(*
SPDX-FileCopyrightText: © 2026 Oleksandr Tiutyk <trofimich@gmail.com>
SPDX-License-Identifier: MIT
License: https://opensource.org/license/mit
*)

(*!
<summary>
Sample activity that steps integer XPosition and YPosition workflow variables toward configured coordinates.
</summary>
<description>
Advances each coordinate by one unit per timer interval until both reach ToXPosition and ToYPosition. Supports
suspension with remaining-time preservation, cancellation, resetting and failure timer cleanup.
</description>
*)

{attribute 'no_explicit_call' := 'do not call this function block directly'}
{attribute 'enable_dynamic_creation'}
FUNCTION_BLOCK MoveFromToActivity EXTENDS TOF_Workflow.Activity IMPLEMENTS IMoveFromToActivity
VAR_STAT
	{attribute 'hide'} 
	_ClassName : STRING := __POUNAME();
END_VAR
VAR
	_ToXPosition : INT;
	_ToYPosition : INT;
	
	_PositionChangeTimer : TOF_Timers.Timer("PositionChangeTimer");
	//! <summary>Time left before the next position step, captured when suspension begins.</summary>
	_RemainingPositionChangeTime : TIME;
END_VAR
VAR CONSTANT
	//! <summary>Delay before the first position step and between subsequent steps; suspended time is excluded.</summary>
	POSITION_CHANGE_TIMER_INTERVAL : TIME := T#10MS;
END_VAR

(*!
<summary>Gets the runtime class name of this object.</summary>
*)
{attribute 'monitoring' := 'call'}
PROPERTY ClassName : REFERENCE TO STRING
GET
ClassName REF= _ClassName;
END_GET
END_PROPERTY

(*!
<summary>Sets the target integer X and Y coordinates for the activity.</summary>
<param name="toXPosition">Target X coordinate.</param>
<param name="toYPosition">Target Y coordinate.</param>
*)
METHOD Configure
VAR_INPUT
	toXPosition : INT;
	toYPosition : INT;
END_VAR
_ToXPosition := toXPosition;
_ToYPosition := toYPosition;
END_METHOD

(*!
<summary>Gets the namespace name of this object.</summary>
*)
{attribute 'monitoring' := 'call'}
PROPERTY NamespaceName : REFERENCE TO STRING
GET
NamespaceName REF= CurrentNamespace.Name;
END_GET
END_PROPERTY

(*!
<summary>Stops the position-change timer and clears saved remaining time when the activity fails.</summary>
<param name="exception">Exception that caused the failure.</param>
*)
METHOD PROTECTED OnFail
VAR_INPUT
	exception : TOF_Core.IException;
END_VAR
_RemainingPositionChangeTime := TOF_Core.Times.MIN_VALUE;

IF _PositionChangeTimer.State.Running THEN
	_PositionChangeTimer.Cancel();
	_PositionChangeTimer.Execute();
END_IF
END_METHOD

(*!
<summary>Stops the position-change timer and clears saved remaining time during resetting.</summary>
<param name="startResetting">TRUE on the initial RequestReset call; FALSE on subsequent Execute cycles.</param>
*)
METHOD PROTECTED OnResetting : TOF_Workflow.ACTIVITY_RESETTING_STATE
VAR_INPUT
	startResetting : BOOL;
END_VAR
_RemainingPositionChangeTime := TOF_Core.Times.MIN_VALUE;

IF _PositionChangeTimer.State.Running THEN
	_PositionChangeTimer.Cancel();
	_PositionChangeTimer.Execute();
END_IF

IF NOT _PositionChangeTimer.State.Running THEN
	OnResetting := TOF_Workflow.ACTIVITY_RESETTING_STATE.WORK_RESET;
END_IF
END_METHOD

(*!
<summary>Moves each coordinate by one unit after each position-change interval.</summary>
<description>
A fresh run restarts the timer with the full interval; resuming restarts it with the remaining time captured
by OnStopping, excluding suspended time. After a resumed step, subsequent steps use the full interval again.
An elapsed interval advances at most one step per call; missed intervals are not replayed. A refused timer
restart returns WORK_HALTED with a diagnostic, preserving any coordinate changes already made. Variable lookup
and conversion exceptions propagate to the activity's failure handling. The activity owner drives these
callbacks sequentially; they do not drive the activity recursively.
</description>
<param name="startRunning">Begins a fresh run, including reuse after an earlier run.</param>
<param name="startResuming">Resumes the remaining interval saved during suspension.</param>
<param name="haltReason">Describes a refused timer restart when WORK_HALTED is returned.</param>
*)
METHOD PROTECTED OnRunning : TOF_Workflow.ACTIVITY_RUNNING_STATE
VAR_INPUT
	startRunning : BOOL;
	startResuming : BOOL;
END_VAR
VAR_OUTPUT
	haltReason : WSTRING(255);
END_VAR
VAR
	xPosition : TOF_Core.GENERIC_VALUE;
	yPosition : TOF_Core.GENERIC_VALUE;

	currentXPosition : INT;
	currentYPosition : INT;
	
END_VAR
IF startRunning THEN
	IF NOT _PositionChangeTimer.SetIntervalAndRestart(interval := POSITION_CHANGE_TIMER_INTERVAL) THEN
		haltReason := "Could not start the position-change timer";
		OnRunning := TOF_Workflow.ACTIVITY_RUNNING_STATE.WORK_HALTED;
	END_IF
ELSIF startResuming THEN
	IF NOT _PositionChangeTimer.SetIntervalAndRestart(interval := _RemainingPositionChangeTime) THEN
		haltReason := "Could not resume the position-change timer";
		OnRunning := TOF_Workflow.ACTIVITY_RUNNING_STATE.WORK_HALTED;
	END_IF
ELSE
	_PositionChangeTimer.Execute();

	IF _PositionChangeTimer.Elapsed THEN
		IF NOT TryGetVariable(name := 'XPosition', variable => xPosition) THEN
			TOF_Workflow.WorkflowExceptions.ThrowWorkflowVariableNotFound(
				sourceNamespaceName := NamespaceName,
				sourceClassName := ClassName,
				sourcePOUName := __POUNAME(),
				sourcePosition := __POSITION(),
				message := "Variable 'XPosition' was not found"
			);
		END_IF
		
		IF NOT TryGetVariable(name := 'YPosition', variable => yPosition) THEN
			TOF_Workflow.WorkflowExceptions.ThrowWorkflowVariableNotFound(
				sourceNamespaceName := NamespaceName,
				sourceClassName := ClassName,
				sourcePOUName := __POUNAME(),
				sourcePosition := __POSITION(),
				message := "Variable 'YPosition' was not found"
			);			
		END_IF
		
		currentXPosition := xPosition.AsInt();
		currentYPosition := yPosition.AsInt();
		
		IF currentXPosition <> _ToXPosition THEN
			IF currentXPosition < _ToXPosition THEN
				currentXPosition := currentXPosition + 1;
			ELSE
				currentXPosition := currentXPosition - 1;
			END_IF
			
			xPosition.ChangeValueByAny(value := currentXPosition);
		END_IF
		
		IF currentYPosition <> _ToYPosition THEN
			IF currentYPosition < _ToYPosition THEN
				currentYPosition := currentYPosition + 1;
			ELSE
				currentYPosition := currentYPosition - 1;
			END_IF
			
			yPosition.ChangeValueByAny(value := currentYPosition);
		END_IF
		
		IF currentXPosition <> _ToXPosition OR_ELSE currentYPosition <> _ToYPosition THEN
			IF NOT _PositionChangeTimer.SetIntervalAndRestart(interval := POSITION_CHANGE_TIMER_INTERVAL) THEN
				haltReason := "Could not restart the position-change timer";
				OnRunning := TOF_Workflow.ACTIVITY_RUNNING_STATE.WORK_HALTED;
			END_IF
		ELSE		
			OnRunning := TOF_Workflow.ACTIVITY_RUNNING_STATE.WORK_COMPLETED;
		END_IF
	END_IF
END_IF
END_METHOD

(*!
<summary>Stops the position-change timer and preserves the remaining interval on suspension.</summary>
<description>
On the first suspension call, updates the timer and saves its remaining interval before cancellation. If the
interval has elapsed, saves zero so the first Execute after resume can perform the pending step. No
coordinates change here. Cancels an active timer and advances stopping; WORK_STOPPED is returned only after it
is no longer running. Further stopping calls preserve the saved remaining time. Exceptions propagate to the
activity's failure handling; captured time and timer effects are not rolled back.
</description>
<param name="startCancelling">
Marks the initial cancellation request; cancellation does not save a resume interval.
</param>
<param name="startSuspending">Marks the initial suspension request and captures the remaining interval once.</param>
<param name="haltReason">No halt diagnostic is produced by ordinary timer stopping.</param>
*)
METHOD PROTECTED OnStopping : TOF_Workflow.ACTIVITY_STOPPING_STATE
VAR_INPUT
	startCancelling : BOOL;
	startSuspending : BOOL;
END_VAR
VAR_OUTPUT
	haltReason : WSTRING(255);
END_VAR
IF startSuspending THEN
	_PositionChangeTimer.Execute();

	IF _PositionChangeTimer.ElapsedTime < _PositionChangeTimer.Interval THEN
		_RemainingPositionChangeTime := _PositionChangeTimer.Interval - _PositionChangeTimer.ElapsedTime;
	ELSE
		_RemainingPositionChangeTime := TOF_Core.Times.MIN_VALUE;
	END_IF
END_IF

IF _PositionChangeTimer.State.Running THEN
	_PositionChangeTimer.Cancel();
	_PositionChangeTimer.Execute();
END_IF

IF NOT _PositionChangeTimer.State.Running THEN
	OnStopping := TOF_Workflow.ACTIVITY_STOPPING_STATE.WORK_STOPPED;
END_IF
END_METHOD

(*!
<summary>Gets the size in bytes of this function block instance.</summary>
*)
{attribute 'monitoring' := 'call'}
PROPERTY SelfSize : ULINT
GET
SelfSize := XSIZEOF(THIS^);
END_GET
END_PROPERTY

(*!
<summary>Gets the configured target X coordinate.</summary>
*)
PROPERTY ToXPosition : INT
GET
ToXPosition := _ToXPosition;
END_GET
END_PROPERTY

(*!
<summary>Gets the configured target Y coordinate.</summary>
*)
PROPERTY ToYPosition : INT
GET
ToYPosition := _ToYPosition;
END_GET
END_PROPERTY

END_FUNCTION_BLOCK

(* stored: Version 1.1.0.1
   POU MoveFromToActivity: Id {3e439478-2975-438e-b7bb-9ad4531af15c}, SpecialFunc None
   Folder Overriden methods: Id {7fdac448-b90e-4952-a44c-a57d67c7342e}
   Property ClassName: Id {a66a843c-b1e9-49fb-b1bd-eb30c1a59478}
   Get Get: Id {684d0e63-ba64-4197-8549-110764775012}
   Method Configure: Id {eac7bd11-88b0-437c-b3da-fdca548034fb}
   Property NamespaceName: Id {e00b0c07-e227-4744-b352-43bc3b73d1fd}
   Get Get: Id {a0c0e8db-f447-4081-a52b-0b41216a5713}
   Method OnFail: Id {b64d892c-3e19-4c87-a520-8f4e2a9c1b73}
   Method OnResetting: Id {c71e49a8-5b20-4f31-9d40-2a6b8e1c5f92}
   Method OnRunning: Id {531b20aa-04ec-447d-8df6-e631e6e7a6ba}
   Method OnStopping: Id {9d74ecb1-a096-400b-ae1c-aa5003999773}
   Property SelfSize: Id {26396f5b-789d-4f77-902f-bac2f3ab39b8}
   Get Get: Id {170a8207-e92a-43d3-98ef-dc6222e69a3d}
   Property ToXPosition: Id {f565365f-3d75-4cc9-9b98-f46d263c2bfe}
   Get Get: Id {766972fc-3f3f-46e2-bcb0-ef52cecd7f9d}
   Property ToYPosition: Id {d3b1e4d2-5064-4089-b170-51f50dc5d7d2}
   Get Get: Id {02f2f180-5bb0-494f-90ce-5e2005e46225} *)
